Universal Robots PolyScope program: TEST_EVAC.urp

Program TEST_EVAC (installation=GD directory=/programs/GD createdIn=5.13.0 lastSavedIn=5.13.0 robotSerialNumber=20205000017)
Calibrated DH parameters: a=[-0.000157, -0.56303, -0.236706, -0.000074, -0.000109, 0]; d=[0.181705, 47.632387, 369.599619, -417.058513, 0.119878, 0.115667]; alpha=[1.570881, -0.005074, -0.001247, 1.56886, -1.570997, 0]; deltaTheta=[0, -0.405485, 5.544791, 1.143886, -0.000009, -0.000001]
InitVariablesNode
BeforeStart
  Script file /programs/GD/CONTROL/ZONE_CONTROL.script
    | def GET_DIST(P1, P2):
    |   return pose_dist(P1, P2)
    | end
    | def CHECK_DIST_NEAR(P1, P2, th):
    |   return (GET_DIST(P1, P2) < th)
    | end
    | def DIST_HOME():
    |   return pose_dist(gHome_Position,CurrPos_p)
    | end
    | 
    | def CHECK_HOME():
    |   return (DIST_HOME()<ZoneDistTh)
    | end
    | 
    | def DIST_CVUpper():
    |   if (read_input_integer_register(4)==1):
    |     p=g2GD_pos1
    |   else:
    |     p=g1GD_pos1
    |   end
    |   return pose_dist(p,CurrPos_p)
    | end
    | 
    | def CHECK_CVUpper():
    |   return (DIST_CVUpper()<ZoneDistTh)
    | end
    | 
    | def CHECK_RB_POS(prg_no):
    |   ret=True
    |   if (prg_no==1001):
    |     ret=CHECK_EVAC()
    |   end
    |   if ((prg_no==1201) or (prg_no==1401) or (prg_no==1402) or (prg_no==6001) or (prg_no==6101) or (prg_no==6401) or (prg_no==6102) or (prg_no==7001)):
    |     ret=CHECK_HOME()
    |   end
    |   if ((prg_no==1002) or (prg_no==1241) or (prg_no==1261)):
    |     ret=CHECK_BKInside()
    |   end
    |   if (prg_no==1251):
    |     ret=(CHECK_HOME() or CHECK_CVUpper())
    |   end
    |   if (ret != True):
    |     SubPrgResult=801
    |     sleep(999999.0)
    |   end
    | end
    | 
    | def DIST_ORIGIN():
    |   p=CurrPos_p
    |   o=p
    |   o[0]=0.0
    |   o[1]=0.0
    |   DistOrigin=pose_dist(o,p)
    |   return pose_dist(o,p)
    | end
    | 
    | def CHECK_EVAC_ORG():
    |   return (EvacRadiusTh<DIST_ORIGIN())
    | end
    | 
    | def CHECK_EVAC_X():
    |   return (EvacXTh[0]<CurrPos_p[0] and CurrPos_p[0]<EvacXTh[1])
    | end
    | 
    | def CHECK_EVAC_Y():
    |   return (EvacYTh[0]<CurrPos_p[1] and CurrPos_p[1]<EvacYTh[1])
    | end
    | 
    | def CHECK_EVAC_Z():
    |   return (EvacZTh[0]<CurrPos_p[2] and CurrPos_p[2]<EvacZTh[1])
    | end
    | 
    | def CHECK_EVAC():
    |   ret=True
    |   ret=(ret and CHECK_EVAC_ORG())
    |   ret=(ret and CHECK_EVAC_X())
    |   ret=(ret and CHECK_EVAC_Y())
    |   ret=(ret and CHECK_EVAC_Z())
    |   return ret
    | end
    | 
    | def CHECK_BKInside():
    |   ret=True
    |   pos=read_input_integer_register(4)
    |   if (pos>2):
    |     ret=False
    |   else:
    |     if (not read_input_boolean_register(13+pos)):
    |       ret=False
    |       ver_3=read_input_boolean_register(13+pos)
    |     else:
    |       bk=pBucket[pos-1]
    |       if (pos==1):
    |         ret=(ret and CurrPos_p[0]>ZoneHomeX)
    |         ret=(ret and bk[1]-(BucketWidth-ZoneBucketGap)<CurrPos_p[1] and CurrPos_p[1]<bk[1]-ZoneBucketGap)
    |       elif (pos==2):
    |         ret=(ret and CurrPos_p[0]<-ZoneHomeX)
    |         ret=(ret and bk[1]+ZoneBucketGap<CurrPos_p[1] and CurrPos_p[1]<bk[1]+(BucketWidth-ZoneBucketGap))
    |       end
    |     end
    |   end
    |   return ret
    | end
    | 
    | def CHECK_CVOutside():
    |   ret=True
    |   ret=(ret and gCV_11_M[0]-Zone6ThX<CurrPos_p[0])
    |   ret=(ret and CurrPos_p[0]<gCV_11_M[0]+Zone6ThX)
    |   ret=(ret and gCV_11_M[1]-Zone6ThY<CurrPos_p[1])
    |   ret=(ret and CurrPos_p[1]<gCV_11_M[1]+Zone6ThY)
    |   return (not ret)
    | end
    | 
    | def CHECK_ZONE(no):
    |   if (no==1):
    |     return (CurrPos_p[2]>=Zone1ZTh)
    |   elif (no==2):
    |     return (CurrPos_p[0]>ZoneHomeX)
    |   elif (no==3):
    |     return (CurrPos_p[0]<-ZoneHomeX)
    |   elif (no==4):
    |     return CHECK_CVUpper()
    |   elif (no==5):
    |     return CHECK_BKInside()
    |   elif (no==6):
    |     return CHECK_CVOutside()
    |   end
    | end
  Set NoAction tcp=TCP_1
Robot Program (runOnlyOnce=true)
  var_1 := False
  If var_1
    MoveL speed 250 mm/s, acceleration 100 mm/s^2 (useActiveTCP=false) tcp=TCP_1; feature=Base
      Waypoint Variable (Variable): variable(featureName=gHome_Position)
      Wait Sleep waitTime=1
      Popup Message (haltProgram=false message=home inputType=Text)
      Waypoint Variable (Variable): variable(featureName=g1GD_pos1)
      Wait Sleep waitTime=1
      Popup Message (haltProgram=false message=pos1 inputType=Text)
      Waypoint Variable (Variable): variable(featureName=g1GD_pos2)
      Wait Sleep waitTime=1
      Popup Message (haltProgram=false message=pos2 inputType=Text)
      Waypoint Variable (Variable): variable(featureName=g1GD_pos3)
      Wait Sleep waitTime=1
      Popup Message (haltProgram=false message=pos3 inputType=Text)
      Waypoint Variable (Variable): variable(featureName=g1GD_pos4)
      Wait Sleep waitTime=1
      Popup Message (haltProgram=false message=pos4 inputType=Text)
      Waypoint Variable (Variable): variable(featureName=g1GD_pos5)
      Wait Sleep waitTime=1
      Popup Message (haltProgram=false message=pos5 inputType=Text)
  Else 
    MoveL speed 250 mm/s, acceleration 100 mm/s^2 (useActiveTCP=false) tcp=TCP_1; feature=Base
      Waypoint Variable (Variable): variable(featureName=g1GD_pos5)
      Wait Sleep waitTime=1
      Popup Message (haltProgram=false message=pos5 inputType=Text)
      Waypoint Variable (Variable): variable(featureName=g1GD_pos4)
      Wait Sleep waitTime=1
      Popup Message (haltProgram=false message=pos4 inputType=Text)
      Waypoint Variable (Variable): variable(featureName=g1GD_pos3)
      Wait Sleep waitTime=1
      Popup Message (haltProgram=false message=pos3 inputType=Text)
      Waypoint Variable (Variable): variable(featureName=g1GD_pos2)
      Wait Sleep waitTime=1
      Popup Message (haltProgram=false message=pos2 inputType=Text)
      Waypoint Variable (Variable): variable(featureName=g1GD_pos1)
      Wait Sleep waitTime=1
      Popup Message (haltProgram=false message=pos1 inputType=Text)
      Waypoint Variable (Variable): variable(featureName=gHome_Position)
      Wait Sleep waitTime=1
      Popup Message (haltProgram=false message=home inputType=Text)
Thread スレッド_2 (runOnlyOnce=false)
  Script: CurrPos=get_actual_tool_flange_pose()
  Script: CurrPos_p=get_actual_tcp_pose()
  Script: Currpos_p_UF0=pose_trans(pose_inv(UF), CurrPos_p)
  TCPSpeed := get_actual_tcp_speed()
  TCPForce := get_tcp_force()
  var_2 := CHECK_EVAC()
  var_3 := CHECK_HOME()
  Script: sync()
